// TIA Portal V20 export
FUNCTION "LER_AxisCtrlCommand" : Void   // FC94, LAD
// stored: Access Published, SetENOAutomatically false
   VAR_INPUT
      enable : Bool;
   END_VAR
   VAR_IN_OUT
      Command : USInt;
      AxisControl : "LBC_typeAxisControlNode";
   END_VAR
   VAR CONSTANT
      CommandReset : USInt;
      CommandMoveVelocity : USInt := 1;
      CommandTorqueLimiting : USInt := 2;
      CommandHoming : USInt := 3;
      CommandPosRelative : USInt := 4;
      CommandposAbsolute : USInt := 5;
      CommandposSuperimposed : USInt := 6;
      CommandHalt : USInt := 7;
      CommandGearIn : USInt := 8;
      CommandCamIn : USInt := 9;
      CommandGearOutCamOut : USInt := 10;
      CommandPhasing : USInt := 11;
   END_VAR
BEGIN

REGION Network 1: Rising edge: Move an axis at constant velocity/speed
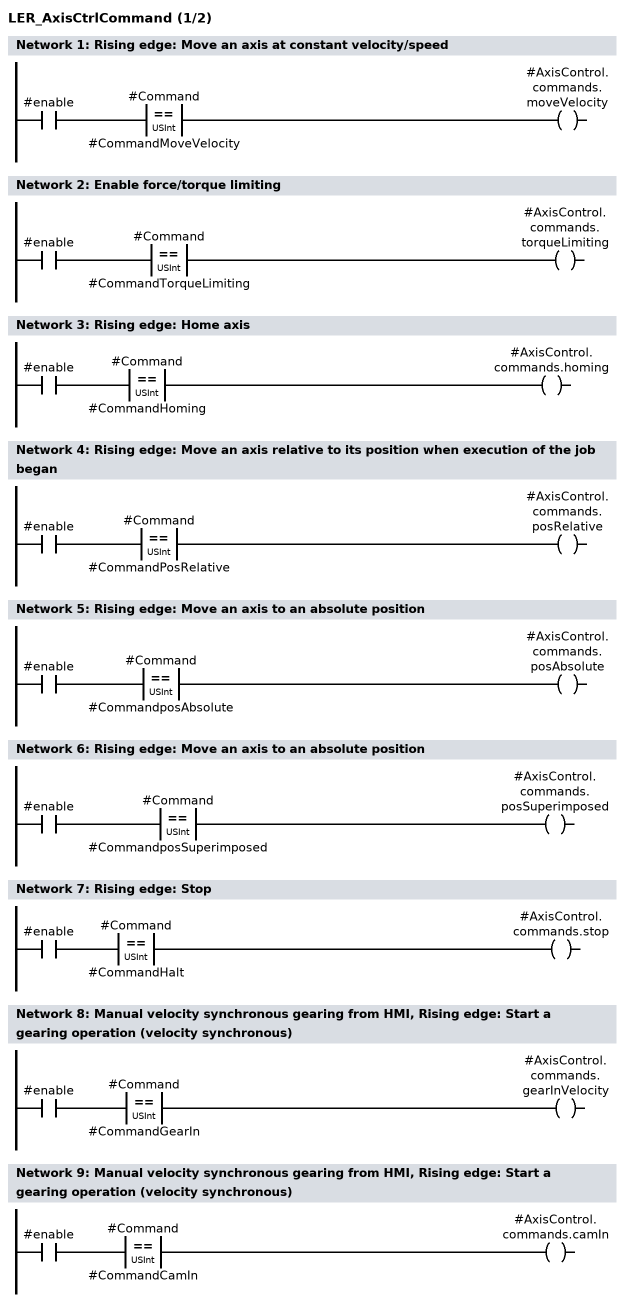
   RUNG wire#powerrail
      Contact( #enable )
      { S7_Templates := "SrcType := USInt" } EQ_Contact(in1 := #Command, in2 := #CommandMoveVelocity)
      Coil( #AxisControl.commands.moveVelocity )
   END_RUNG
   // the same network as SCL:
   #AxisControl.commands.moveVelocity := #enable AND (#Command = #CommandMoveVelocity);
END_REGION

REGION Network 2: Enable force/torque limiting
   RUNG wire#powerrail
      Contact( #enable )
      { S7_Templates := "SrcType := USInt" } EQ_Contact(in1 := #Command, in2 := #CommandTorqueLimiting)
      Coil( #AxisControl.commands.torqueLimiting )
   END_RUNG
   // the same network as SCL:
   #AxisControl.commands.torqueLimiting := #enable AND (#Command = #CommandTorqueLimiting);
END_REGION

REGION Network 3: Rising edge: Home axis
   RUNG wire#powerrail
      Contact( #enable )
      { S7_Templates := "SrcType := USInt" } EQ_Contact(in1 := #Command, in2 := #CommandHoming)
      Coil( #AxisControl.commands.homing )
   END_RUNG
   // the same network as SCL:
   #AxisControl.commands.homing := #enable AND (#Command = #CommandHoming);
END_REGION

REGION Network 4: Rising edge: Move an axis relative to its position when execution of the job began
   RUNG wire#powerrail
      Contact( #enable )
      { S7_Templates := "SrcType := USInt" } EQ_Contact(in1 := #Command, in2 := #CommandPosRelative)
      Coil( #AxisControl.commands.posRelative )
   END_RUNG
   // the same network as SCL:
   #AxisControl.commands.posRelative := #enable AND (#Command = #CommandPosRelative);
END_REGION

REGION Network 5: Rising edge: Move an axis to an absolute position
   RUNG wire#powerrail
      Contact( #enable )
      { S7_Templates := "SrcType := USInt" } EQ_Contact(in1 := #Command, in2 := #CommandposAbsolute)
      Coil( #AxisControl.commands.posAbsolute )
   END_RUNG
   // the same network as SCL:
   #AxisControl.commands.posAbsolute := #enable AND (#Command = #CommandposAbsolute);
END_REGION

REGION Network 6: Rising edge: Move an axis to an absolute position
   RUNG wire#powerrail
      Contact( #enable )
      { S7_Templates := "SrcType := USInt" } EQ_Contact(in1 := #Command, in2 := #CommandposSuperimposed)
      Coil( #AxisControl.commands.posSuperimposed )
   END_RUNG
   // the same network as SCL:
   #AxisControl.commands.posSuperimposed := #enable AND (#Command = #CommandposSuperimposed);
END_REGION

REGION Network 7: Rising edge: Stop
   RUNG wire#powerrail
      Contact( #enable )
      { S7_Templates := "SrcType := USInt" } EQ_Contact(in1 := #Command, in2 := #CommandHalt)
      Coil( #AxisControl.commands.stop )
   END_RUNG
   // the same network as SCL:
   #AxisControl.commands.stop := #enable AND (#Command = #CommandHalt);
END_REGION

REGION Network 8: Manual velocity synchronous gearing from HMI, Rising edge: Start a gearing operation (velocity synchronous)
   RUNG wire#powerrail
      Contact( #enable )
      { S7_Templates := "SrcType := USInt" } EQ_Contact(in1 := #Command, in2 := #CommandGearIn)
      Coil( #AxisControl.commands.gearInVelocity )
   END_RUNG
   // the same network as SCL:
   #AxisControl.commands.gearInVelocity := #enable AND (#Command = #CommandGearIn);
END_REGION

REGION Network 9: Manual velocity synchronous gearing from HMI, Rising edge: Start a gearing operation (velocity synchronous)
   RUNG wire#powerrail
      Contact( #enable )
      { S7_Templates := "SrcType := USInt" } EQ_Contact(in1 := #Command, in2 := #CommandCamIn)
      Coil( #AxisControl.commands.camIn )
   END_RUNG
   // the same network as SCL:
   #AxisControl.commands.camIn := #enable AND (#Command = #CommandCamIn);
END_REGION

REGION Network 10
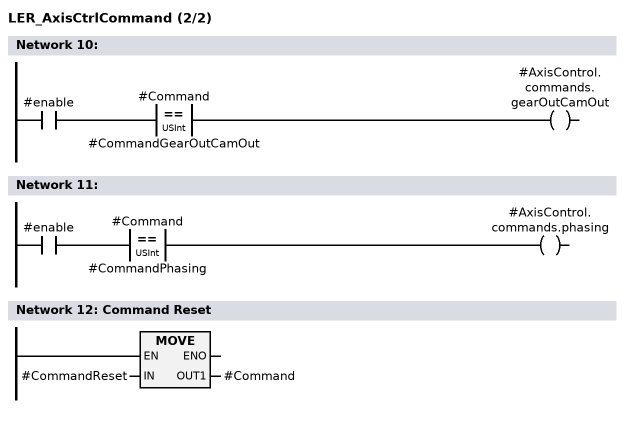
   RUNG wire#powerrail
      Contact( #enable )
      { S7_Templates := "SrcType := USInt" } EQ_Contact(in1 := #Command, in2 := #CommandGearOutCamOut)
      Coil( #AxisControl.commands.gearOutCamOut )
   END_RUNG
   // the same network as SCL:
   #AxisControl.commands.gearOutCamOut := #enable AND (#Command = #CommandGearOutCamOut);
END_REGION

REGION Network 11
   RUNG wire#powerrail
      Contact( #enable )
      { S7_Templates := "SrcType := USInt" } EQ_Contact(in1 := #Command, in2 := #CommandPhasing)
      Coil( #AxisControl.commands.phasing )
   END_RUNG
   // the same network as SCL:
   #AxisControl.commands.phasing := #enable AND (#Command = #CommandPhasing);
END_REGION

REGION Network 12: Command Reset
   RUNG wire#powerrail
      Move(in := #CommandReset, out1 => #Command)
   END_RUNG
   // the same network as SCL:
   #Command := #CommandReset;
END_REGION
END_FUNCTION
